(* CoDeSys 2.3 library: TcModbusSrv.lib *)
(* Libraries: STANDARD.LIB 5.6.98 11:03:02, TcBase.lib 14.5.09 11:14:08, TcSystem.lib 18.2.11 16:15:48 *)

(* Global variable list: Globale_Variablen *)
VAR_GLOBAL CONSTANT
	AMSPORT_R3_MODBUSSERV		:	UINT:= 10500;
	MODBUS_TCP_PORT				: 	UINT := 502;
	MB_MAXSIZE					: 	UDINT:= 260;
	MBADS_IGR_CLOSEALL			:	UDINT:=16#00001001;
	MBADS_IGR_UDP_FLAG			:	DWORD:=16#80000000;
END_VAR

(* Data type *)
TYPE E_MBFctCodes :						(*Modbus Function Codes*)
(
	MBFCT_READCOILS:=1,				(*Read Multiple Output Coils*)
	MBFCT_READINPUTS:=2	,			(*Read Multiple Input Coils*)
	MBFCT_READREGISTERS := 3,			(*Read Multiple Output Registers*)
	MBFCT_READINPUTREGISTERS:=4, 	(*Read Multiple Input Registers*)
	MBFCT_WRITESINGLECOIL:=5,
	MBFCT_WRITESINGLEREGISTER:= 6,
	MBFCT_DIAGNOSE:=8,
	MBFCT_WRITECOILS:=15,
	MBFCT_WRITEREGISTERS := 16,		(* Write Multiple Registers*)
	MBFCT_READWRITEREGISTERS := 23
);
END_TYPE

(* Data type *)
TYPE ST_MBAddr :
STRUCT
	arrIpAddr	: ARRAY[0..3] OF BYTE;
	nPort		: UINT;
	nUnitId		: BYTE;
END_STRUCT
END_TYPE

(* Data type *)
TYPE ST_MBReadWrite :
STRUCT
	arrIpAddr	: ARRAY[0..3]  OF BYTE;
	nPort		: UINT;
	nUnitId		: BYTE;
	nStartAddr	: ARRAY[0..1] OF BYTE;
	nQuantity	: ARRAY[0..1] OF BYTE;
	arrBuffer	: ARRAY [1..MB_MAXSIZE] OF BYTE;
	dummy	: BYTE;(* not used *)
END_STRUCT
END_TYPE

(* Data type *)
TYPE ST_MBWrite :
STRUCT
	arrIpAddr	: ARRAY[0..3]  OF BYTE;
	nPort		: UINT;
	nUnitId		: BYTE;
	arrBuffer	: ARRAY[1..MB_MAXSIZE] OF BYTE;
	dummy	: BYTE;(* not used *)
END_STRUCT
END_TYPE

(* Data type *)
TYPE ST_MBWriteSingle :
STRUCT
	arrIpAddr	: ARRAY [0..3]  OF BYTE;
	nPort		: UINT;
	nUnitId		: BYTE;
	nValue 	: ARRAY[0..1] OF BYTE;
END_STRUCT
END_TYPE

(* POU F_GetIPAddrFromStr, ST *)
FUNCTION F_GetIPAddrFromStr: ARRAY[0..3] OF BYTE
VAR_INPUT
	sIPAddr	: STRING(15);
END_VAR
VAR
	pIp		: POINTER TO BYTE;
	b		: ARRAY[0..3] OF BYTE;
	w		: WORD;
	id		: INT;
END_VAR
pIp := ADR( sIpAddr );
id 		:= 0;
w		:= 0;

WHILE pIp^ <> 0 DO
	CASE pIp^ OF
		16#30..16#39: (* Numbers 0..9 *)
			w := ( w * 10 ) + ( pIp^ - 16#30 );
			IF w <= 255 THEN
				b[id] := WORD_TO_BYTE( w );
			ELSE
				RETURN; (* number overflow *)
			END_IF
		16#2E: (* dot *)
			IF id < 3 THEN
				w		:= 0;	(* reset temp variable *)
				id 		:= id + 1;	(* increment to the next id *)
			ELSE
				RETURN; (* to many numbers *)
			END_IF
	ELSE
		RETURN; (* unresolved characters *)
	END_CASE
	pIp := pIp + 1;
END_WHILE

(* check the number of scanned numbers again *)
IF ( id = 0 ) OR ( id = 3 ) THEN
	F_GetIPAddrFromStr := b; (* OK *)
ELSE
	RETURN; (* error, not all ids scanned! *)
END_IF
END_FUNCTION

(* POU F_GetVersionTcModbusSrv, ST *)
FUNCTION F_GetVersionTcModbusSrv : UINT
(* Returns the library version information  *)
VAR_INPUT
       nVersionElement       :       INT;
END_VAR
VAR
END_VAR 
(* Version history:
Date [DD.MM.YYYY]	| Version    		| created under      			| Author         		| Remark 
------------------------------------------------------------------------------------------------------------------------------------------------------ 
26.10.2005    			| 1.0.1      			| V2.10.0 (Build 1242) 		| RichardK 		| first release 
07.12.2006			| 1.0.2				| V2.10.0 (Build 1302) 		| RichardK 		| support for arm platforms added
20.02.2008			| 1.0.3				| V2.10.0 (Build 1320) 		| RichardK 		| optimization of F_GetIPAddrFromStr
03.05.2008			| 1.0.4				| V2.10.0 (Build 1323) 		| RichardK 		| init ads functionblocks
15.06.2010			| 1.0.5				| V2.10.0 (Build 1323) 		| RichardK 		| improved perfomance
30.05.2011			| 1.0.6				| V2.10.0 (Build 2029) saved as TwinCAT 2.8 lib	| ChristophC 		| internal used functions and data types moved to [internal used] folder, improved performance, cbRead-output fix
06.12.2011			| 1.0.7				| V2.11.0 (Build 2206)  saved as TwinCAT 2.8 lib	| RichardK 		| added FB_MBCloseAllConnections
11.12.2012			| 1.0.8				| V2.11.0 (Build 2206)  saved as TwinCAT 2.8 lib	| RichardK 		| added udp function blocks
*) 
CASE nVersionElement OF
1: (* major number *)
        F_GetVersionTcModbusSrv := 1;
2: (* minor number *)
       F_GetVersionTcModbusSrv := 0;
3: (* revision number *)
        F_GetVersionTcModbusSrv := 6;
ELSE
   F_GetVersionTcModbusSrv := 16#FFFF;
END_CASE
END_FUNCTION

(* POU FB_MBCloseAll, ST *)
FUNCTION_BLOCK FB_MBCloseAll
VAR_INPUT
	bExecute			: BOOL;(* Rising edge at this input starts command execution *)
	tTimeout			: TIME:=T#1s;
END_VAR
VAR_OUTPUT
	bBusy				: BOOL;
	bError				: BOOL;
	nErrId				: UDINT;
END_VAR
{library private}
VAR
	state 			: UDINT;
	RisingEdge		: R_TRIG;
	fbAdsWrite		: ADSWRITE := ( NETID := '', PORT := AMSPORT_R3_MODBUSSERV, IDXGRP := MBADS_IGR_CLOSEALL );
	cbWLen			: UDINT;
END_VAR
RisingEdge( CLK:= bExecute );
CASE state OF
	0:
		IF RisingEdge.Q THEN
			(* reset outputs *)
			bBusy := TRUE;
			bError := FALSE;
			nErrId := 0;

			fbAdsWrite( IDXOFFS := 0, LEN := 0, SRCADDR :=0,  WRITE := TRUE, TMOUT := tTimeout );
			(* go to the wait state *)
			state := 1;
		END_IF
	1:(* wait until fb not busy *)
		fbAdsWrite( WRITE := FALSE, BUSY=>bBusy, ERR=>bError, ERRID=>nErrID );
		IF NOT fbAdsWrite.BUSY THEN
			state := 0;
		END_IF
END_CASE
END_FUNCTION_BLOCK

(* POU FB_MBDiagnose, ST *)
FUNCTION_BLOCK FB_MBDiagnose
(* Executes diagnostic function *)
VAR_INPUT
	sIPAddr	 		: STRING(15);(* IPv4 address of the target device *)
	nTCPPort			: UINT:= MODBUS_TCP_PORT;(* Port number of the target device *)
	nUnitID			: BYTE:=16#FF;(* Identification number of a serial sub-network device *)
	nSubFnc			: WORD;
	nWriteData		: WORD;
	bExecute			: BOOL;(* Rising edge at this input starts command execution *)
	tTimeout			: TIME:=T#1s;
END_VAR
VAR_OUTPUT
	bBusy				: BOOL;
	bError				: BOOL;
	nErrId				: UDINT;
	nReadData		: WORD;
END_VAR
{library private}
VAR
	state 				: UDINT;
	RisingEdge		: R_TRIG;
	fbAdsRDWRT		: ADSRDWRT := ( NETID := '', PORT := AMSPORT_R3_MODBUSSERV, IDXGRP := MBFCT_DIAGNOSE );
	stMBAddr			: ST_MBAddr;
END_VAR
RisingEdge( CLK:= bExecute );
CASE state OF
	0:
		IF RisingEdge.Q THEN
			(* reset outputs *)
			bBusy := TRUE;
			bError := FALSE;
			nErrId := 0;
			nReadData := 0;
			(* prepare request params *)
			stMBAddr.nPort := nTCPPort;
			stMBAddr.nUnitId := nUnitID;
			stMBAddr.arrIpAddr := F_GetIPAddrFromStr( sIPAddr );
			(* reset fb *)
			fbAdsRDWRT( WRTRD := FALSE );
			(* start command execution *)
			fbAdsRDWRT( IDXOFFS := DWORD_TO_UDINT( SHL( WORD_TO_DWORD( nSubFnc ), 16 ) OR nWriteData  ),
							WRITELEN := SIZEOF( stMBAddr.arrIpAddr ) + SIZEOF( stMBAddr.nPort ) + SIZEOF( stMBAddr.nUnitId ),
							SRCADDR := ADR( stMBAddr ),
							READLEN := SIZEOF( nReadData ),
							DESTADDR := ADR( nReadData ),
							WRTRD := TRUE, TMOUT := tTimeout  );
			(* go to the wait state *)
			state := 1;
		END_IF
	1:(* wait until fb not busy *)
		fbAdsRDWRT( WRTRD := FALSE, BUSY=>bBusy, ERR=>bError, ERRID=>nErrID );
		IF NOT fbAdsRDWRT.BUSY THEN
			state := 0;
		END_IF
END_CASE
END_FUNCTION_BLOCK

(* POU FB_MBReadCoils, ST *)
FUNCTION_BLOCK FB_MBReadCoils
(* Read 1..2048 digital outputs (coils, bit access) *)
VAR_INPUT
	sIPAddr	 		: STRING(15);(* IPv4 address of the target device *)
	nTCPPort			: UINT:= MODBUS_TCP_PORT;(* Port number of the target device *)
	nUnitID			: BYTE:=16#FF;(* Identification number of a serial sub-network device *)
	nQuantity			: WORD;(* Number of coils to read (data bits) *)
	nMBAddr			: WORD;(* Address of start coil (data bit offset) *)
	cbLength			: UDINT;(* Max. byte size of destination buffer *)
	pDestAddr			: UDINT;(* Pointer to destination buffer *)
	bExecute			: BOOL;(* Rising edge at this input starts command execution *)
	tTimeout			: TIME:=T#1s;
END_VAR
VAR_OUTPUT
	bBusy				: BOOL;
	bError				: BOOL;
	nErrId				: UDINT;
	cbRead			: UDINT;
END_VAR
{library private}
VAR
	state 				: UDINT;
	RisingEdge		: R_TRIG;
	fbAdsRDWRT		: ADSRDWRTEX := ( NETID := '', PORT := AMSPORT_R3_MODBUSSERV, IDXGRP := MBFCT_READCOILS );
	stMBAddr			: ST_MBAddr;
	cbRLen			: UDINT;
END_VAR
RisingEdge( CLK:= bExecute );
CASE state OF
	0:
		IF RisingEdge.Q THEN
			(* reset outputs *)
			bBusy := TRUE;
			bError := FALSE;
			nErrId := 0;
			cbRead := 0;
			(* calculate the required target buffer size *)
			cbRLen := ( nQuantity + 7 ) / 8;
			(* check target buffer length *)
			IF( cbRLen <= cbLength ) THEN
				(* prepare request params *)
				stMBAddr.nPort := nTCPPort;
				stMBAddr.nUnitId := nUnitID;
				stMBAddr.arrIpAddr := F_GetIPAddrFromStr( sIPAddr );
				(* reset fb *)
				fbAdsRDWRT( WRTRD := FALSE );
				(* start command execution *)
				fbAdsRDWRT( IDXOFFS := DWORD_TO_UDINT( SHL( WORD_TO_DWORD(nMBAddr), 16 ) OR nQuantity ),
								WRITELEN := SIZEOF( stMBAddr.arrIpAddr ) + SIZEOF( stMBAddr.nPort ) + SIZEOF( stMBAddr.nUnitId ),
								SRCADDR := ADR( stMBAddr ),
								READLEN := cbRLen, DESTADDR := pDestAddr,
								WRTRD := TRUE,	TMOUT := tTimeout );
				(* go to the wait state *)
				state := 1;
			ELSE
				bBusy := FALSE;
				bError:= TRUE;
				nErrId := 16#702;
			END_IF
		END_IF
	1:(* wait until fb not busy *)
		fbAdsRDWRT( WRTRD := FALSE, BUSY=>bBusy, ERR=>bError, ERRID=>nErrID, COUNT_R=>cbRead );
		IF NOT fbAdsRDWRT.BUSY THEN
			state := 0;
		END_IF
END_CASE
END_FUNCTION_BLOCK

(* POU FB_MBReadInputRegs, ST *)
FUNCTION_BLOCK FB_MBReadInputRegs
(* Read 1..128 digital input registers (word access) *)
VAR_INPUT
	sIPAddr	 		: STRING(15);(* IPv4 address of the target device *)
	nTCPPort			: UINT:= MODBUS_TCP_PORT;(* Port number of the target device *)
	nUnitID			: BYTE:=16#FF;(* Identification number of a serial sub-network device *)
	nQuantity			: WORD;(* Number of input registers to read (data words) *)
	nMBAddr			: WORD;(* Address of start input register (data word offset) *)
	cbLength			: UDINT;(* Max. byte size of destination buffer *)
	pDestAddr			: UDINT;(* Pointer to destination buffer *)
	bExecute			: BOOL;(* Rising edge at this input starts command execution *)
	tTimeout			: TIME:=T#1s;
END_VAR
VAR_OUTPUT
	bBusy				: BOOL;
	bError				: BOOL;
	nErrId				: UDINT;
	cbRead			: UDINT;
END_VAR
{library private}
VAR
	state 				: UDINT;
	RisingEdge		: R_TRIG;
	fbAdsRDWRT		: ADSRDWRTEX := ( NETID := '', PORT := AMSPORT_R3_MODBUSSERV, IDXGRP := MBFCT_READINPUTREGISTERS );
	stMBAddr			: ST_MBAddr;
	cbRLen			: UDINT;
END_VAR
RisingEdge( CLK:= bExecute );
CASE state OF
	0:
		IF RisingEdge.Q THEN
			(* reset outputs *)
			bBusy := TRUE;
			bError := FALSE;
			nErrId := 0;
			cbRead := 0;
			(* calculate the required target buffer size *)
			cbRLen := nQuantity * 2;
			(* check target buffer length *)
			IF( cbRLen <= cbLength ) THEN
				(* prepare request params *)
				stMBAddr.nPort := nTCPPort;
				stMBAddr.nUnitId := nUnitID;
				stMBAddr.arrIpAddr := F_GetIPAddrFromStr( sIPAddr );
				(* reset fb *)
				fbAdsRDWRT( WRTRD := FALSE );
				(* start command execution *)
				fbAdsRDWRT( IDXOFFS := DWORD_TO_UDINT( SHL( WORD_TO_DWORD( nMBAddr ), 16 ) OR nQuantity ),
								WRITELEN := SIZEOF( stMBAddr.arrIpAddr ) + SIZEOF( stMBAddr.nPort ) + SIZEOF( stMBAddr.nUnitId ),
								SRCADDR := ADR( stMBAddr ),
								READLEN := cbRLen, DESTADDR := pDestAddr,
								WRTRD := TRUE, TMOUT := tTimeout );
				(* go to the wait state *)
				state := 1;
			ELSE
				bBusy := FALSE;
				bError:= TRUE;
				nErrId := 16#702;
			END_IF
		END_IF
	1:(* wait until fb not busy *)
		fbAdsRDWRT( WRTRD := FALSE, BUSY=>bBusy, ERR=>bError, ERRID=>nErrID, COUNT_R=>cbRead );
		IF NOT fbAdsRDWRT.BUSY THEN
			state := 0;
		END_IF
END_CASE
END_FUNCTION_BLOCK

(* POU FB_MBReadInputs, ST *)
FUNCTION_BLOCK FB_MBReadInputs
(* Read 1..2048 digital inputs (bit access) *)
VAR_INPUT
	sIPAddr	 		: STRING(15);(* IPv4 address of the target device *)
	nTCPPort			: UINT:= MODBUS_TCP_PORT;(* Port number of the target device *)
	nUnitID			: BYTE:=16#FF;(* Identification number of a serial sub-network device *)
	nQuantity			: WORD;(* Number of inputs to read (data bits) *)
	nMBAddr			: WORD;(* Address of start input (data bit offset) *)
	cbLength			: UDINT;(* Max. byte size of destination buffer *)
	pDestAddr			: UDINT;(* Pointer to destination buffer *)
	bExecute			: BOOL;(* Rising edge at this input starts command execution *)
	tTimeout			: TIME:=T#1s;
END_VAR
VAR_OUTPUT
	bBusy				: BOOL;
	bError				: BOOL;
	nErrId				: UDINT;
	cbRead			: UDINT;
END_VAR
{library private}
VAR
	state 				: UDINT;
	RisingEdge		: R_TRIG;
	fbAdsRDWRT		: ADSRDWRTEX := ( NETID := '', PORT := AMSPORT_R3_MODBUSSERV, IDXGRP := MBFCT_READINPUTS );
	stMBAddr			: ST_MBAddr;
	cbRLen			: UDINT;
END_VAR
RisingEdge( CLK:= bExecute );
CASE state OF
	0:
		IF RisingEdge.Q THEN
			(* reset outputs *)
			bBusy := TRUE;
			bError := FALSE;
			nErrId := 0;
			cbRead := 0;
			(* calculate the required target buffer size *)
			cbRLen := ( nQuantity + 7 ) / 8;
			(* check target buffer length *)
			IF( cbRLen <= cbLength ) THEN
				(* prepare request params *)
				stMBAddr.nPort := nTCPPort;
				stMBAddr.nUnitId := nUnitID;
				stMBAddr.arrIpAddr := F_GetIPAddrFromStr( sIPAddr );
				(* reset fb *)
				fbAdsRDWRT( WRTRD := FALSE );
				(* start command execution *)
				fbAdsRDWRT( IDXOFFS := DWORD_TO_UDINT( SHL( WORD_TO_DWORD( nMBAddr ), 16 ) OR nQuantity ),
								WRITELEN := SIZEOF( stMBAddr.arrIpAddr ) + SIZEOF( stMBAddr.nPort )+ SIZEOF( stMBAddr.nUnitId ),
								SRCADDR := ADR( stMBAddr ),
								READLEN := cbRLen, DESTADDR := pDestAddr,
								WRTRD := TRUE, TMOUT := tTimeout );
				(* go to the wait state *)
				state := 1;
			ELSE
				bBusy := FALSE;
				bError:= TRUE;
				nErrId := 16#702;
			END_IF
		END_IF
	1:(* wait until fb not busy *)
		fbAdsRDWRT( WRTRD := FALSE, BUSY=>bBusy, ERR=>bError, ERRID=>nErrID, COUNT_R=>cbRead );
		IF NOT fbAdsRDWRT.BUSY THEN
			state := 0;
		END_IF
END_CASE
END_FUNCTION_BLOCK

(* POU FB_MBReadRegs, ST *)
FUNCTION_BLOCK FB_MBReadRegs
(* Read 1..128 output registers (word access) *)
VAR_INPUT
	sIPAddr	 		: STRING(15);(* IPv4 address of the target device *)
	nTCPPort			: UINT:= MODBUS_TCP_PORT;(* Port number of the target device *)
	nUnitID			: BYTE:=16#FF;(* Identification number of a serial sub-network device *)
	nQuantity			: WORD;(* Number of registers to read (data words) *)
	nMBAddr			: WORD;(* Address of start register (data word offset) *)
	cbLength			: UDINT;(* Max. byte size of destination buffer *)
	pDestAddr			: UDINT;(* Pointer to destination buffer *)
	bExecute			: BOOL;(* Rising edge at this input starts command execution *)
	tTimeout			: TIME:=T#1s;
END_VAR
VAR_OUTPUT
	bBusy				: BOOL;
	bError				: BOOL;
	nErrId				: UDINT;
	cbRead			: UDINT;
END_VAR
{library private}
VAR
	state 				: UDINT;
	RisingEdge		: R_TRIG;
	fbAdsRDWRT		: ADSRDWRTEX := ( NETID := '', PORT := AMSPORT_R3_MODBUSSERV, IDXGRP := MBFCT_READREGISTERS );
	stMBAddr			: ST_MBAddr;
	cbRLen			: UDINT;
END_VAR
RisingEdge( CLK:= bExecute );
CASE state OF
	0:
		IF RisingEdge.Q THEN
			(* reset outputs *)
			bBusy := TRUE;
			bError := FALSE;
			nErrId := 0;
			cbRead := 0;
			(* calculate the required target buffer size *)
			cbRLen := nQuantity * 2;
			(* check target buffer length *)
			IF( cbRLen <= cbLength ) THEN
				(* prepare request params *)
				stMBAddr.nPort := nTCPPort;
				stMBAddr.nUnitId := nUnitID;
				stMBAddr.arrIpAddr := F_GetIPAddrFromStr( sIPAddr );
				(* reset fb *)
				fbAdsRDWRT( WRTRD := FALSE );
				(* start command execution *)
				fbAdsRDWRT( IDXOFFS := DWORD_TO_UDINT(  SHL( WORD_TO_DWORD( nMBAddr ), 16 ) OR nQuantity  ),
								WRITELEN := SIZEOF( stMBAddr.arrIpAddr ) + SIZEOF( stMBAddr.nPort ) + SIZEOF( stMBAddr.nUnitId ),
								SRCADDR := ADR( stMBAddr ),
								READLEN := cbRLen, DESTADDR := pDestAddr,
								WRTRD := TRUE, TMOUT := tTimeout );
				(* go to the wait state *)
				state := 1;
			ELSE
				bBusy := FALSE;
				bError:= TRUE;
				nErrId := 16#702;
			END_IF
		END_IF
	1:(* wait until fb not busy *)
		fbAdsRDWRT( WRTRD := FALSE, BUSY=>bBusy, ERR=>bError, ERRID=>nErrID, COUNT_R=>cbRead );
		IF NOT fbAdsRDWRT.BUSY THEN
			state:= 0;
		END_IF
END_CASE
END_FUNCTION_BLOCK

(* POU FB_MBReadWriteRegs, ST *)
FUNCTION_BLOCK FB_MBReadWriteRegs
(* Reads 1..128 output registers and writes 1..128 output registers (word access) *)
VAR_INPUT
	sIPAddr	 		: STRING(15);(* IPv4 address of the target device *)
	nTCPPort			: UINT:= MODBUS_TCP_PORT;(* Port number of the target device *)
	nUnitID			: BYTE:=16#FF;(* Identification number of a serial sub-network device *)
	nReadQuantity	: WORD;(* Number of registers to read (data words) *)
	nMBReadAddr		: WORD;(* Address of start read register (data word offset) *)
	nWriteQuantity		: WORD;(* Number of registers to write (data words) *)
	nMBWriteAddr		: WORD;(* Address of start write register (data word offset) *)
	cbDestLength		: UDINT;(* Max. byte size of destination buffer *)
	pDestAddr			: UDINT;(* Pointer to destination buffer *)
	cbSrcLength		: UDINT;(* Max. byte size of source buffer *)
	pSrcAddr			: UDINT;(* Pointer to source buffer *)
	bExecute			: BOOL;(* Rising edge at this input starts command execution *)
	tTimeout			: TIME:=T#1s;
END_VAR
VAR_OUTPUT
	bBusy				: BOOL;
	bError				: BOOL;
	nErrId				: UDINT;
	cbRead			: UDINT;
END_VAR
{library private}
VAR
	state 				: UDINT;
	RisingEdge		: R_TRIG;
	fbAdsRDWRT		: ADSRDWRTEX := ( NETID := '', PORT := AMSPORT_R3_MODBUSSERV, IDXGRP := MBFCT_READWRITEREGISTERS );
	stMBReadWrite	: ST_MBReadWrite;
	cbRLen			: UDINT;
	cbWLen			: UDINT;
END_VAR
RisingEdge( CLK:= bExecute );
CASE state OF
	0:
		IF RisingEdge.Q THEN
			(* reset outputs *)
			bBusy := TRUE;
			bError := FALSE;
			nErrId := 0;
			cbRead := 0;
			(* calculate the required source and target buffer byte size *)
			cbRLen   := nReadQuantity * 2;
			cbWLen := nWriteQuantity * 2;
			(* check source and target buffer length *)
			IF( cbRLen <= cbDestLength ) AND ( cbWLen <= cbSrcLength ) AND ( cbWLen <= SIZEOF( stMBReadWrite.arrBuffer ) ) THEN
				(* prepare request params *)
				stMBReadWrite.arrIpAddr := F_GetIPAddrFromStr( sIPAddr );
				stMBReadWrite.nPort := nTCPPort;
				stMBReadWrite.nUnitId := nUnitID;
				(* copy write params to temp buffer *)
				MEMCPY( ADR( stMBReadWrite.nStartAddr ), ADR( nMBWriteAddr ), SIZEOF( stMBReadWrite.nStartAddr ) );
				MEMCPY( ADR( stMBReadWrite.nQuantity ), ADR( nWriteQuantity ), SIZEOF( stMBReadWrite.nQuantity ) );
				MEMCPY( ADR( stMBReadWrite.arrBuffer ), pSrcAddr, cbWLen );
				(* reset fb *)
				fbAdsRDWRT( WRTRD := FALSE );
				(* start command execution *)
				fbAdsRDWRT( IDXOFFS := DWORD_TO_UDINT(  SHL( WORD_TO_DWORD( nMBReadAddr ), 16 ) OR nReadQuantity ),
								WRITELEN := cbWLen + SIZEOF( stMBReadWrite.arrIpAddr ) + SIZEOF( stMBReadWrite.nPort ) + SIZEOF( stMBReadWrite.nUnitId ) + SIZEOF( stMBReadWrite.nStartAddr ) + SIZEOF( stMBReadWrite.nQuantity ),
								SRCADDR := ADR( stMBReadWrite ),
								READLEN := cbRLen, DESTADDR := pDestAddr,
								WRTRD := TRUE,	TMOUT := tTimeout );
				(* go to the wait state *)
				state := 1;
			ELSE
				bBusy := FALSE;
				bError:= TRUE;
				nErrId := 16#702;
			END_IF
		END_IF
	1:(* wait until fb not busy *)
		fbAdsRDWRT( WRTRD := FALSE, BUSY=>bBusy, ERR=>bError, ERRID=>nErrID, COUNT_R=>cbRead );
		IF NOT fbAdsRDWRT.BUSY THEN
			state := 0;
		END_IF
END_CASE
END_FUNCTION_BLOCK

(* POU FB_MBUdpDiagnose, ST *)
FUNCTION_BLOCK FB_MBUdpDiagnose
(* Executes diagnostic function *)
VAR_INPUT
	sIPAddr	 		: STRING(15);(* IPv4 address of the target device *)
	nTCPPort			: UINT:= MODBUS_TCP_PORT;(* Port number of the target device *)
	nUnitID			: BYTE:=16#FF;(* Identification number of a serial sub-network device *)
	nSubFnc			: WORD;
	nWriteData		: WORD;
	bExecute			: BOOL;(* Rising edge at this input starts command execution *)
	tTimeout			: TIME:=T#1s;
END_VAR
VAR_OUTPUT
	bBusy				: BOOL;
	bError				: BOOL;
	nErrId				: UDINT;
	nReadData		: WORD;
END_VAR
{library private}
VAR
	state 				: UDINT;
	RisingEdge		: R_TRIG;
	fbAdsRDWRT		: ADSRDWRT := ( NETID := '', PORT := AMSPORT_R3_MODBUSSERV );
	stMBAddr			: ST_MBAddr;
END_VAR
RisingEdge( CLK:= bExecute );
CASE state OF
	0:
		IF RisingEdge.Q THEN
			(* reset outputs *)
			bBusy := TRUE;
			bError := FALSE;
			nErrId := 0;
			nReadData := 0;
			(* prepare request params *)
			stMBAddr.nPort := nTCPPort;
			stMBAddr.nUnitId := nUnitID;
			stMBAddr.arrIpAddr := F_GetIPAddrFromStr( sIPAddr );
			(* reset fb *)
			fbAdsRDWRT( WRTRD := FALSE );
			(* start command execution *)
			fbAdsRDWRT( IDXGRP :=  DWORD_TO_UDINT(INT_TO_DWORD(MBFCT_DIAGNOSE) OR MBADS_IGR_UDP_FLAG),
							IDXOFFS := DWORD_TO_UDINT( SHL( WORD_TO_DWORD( nSubFnc ), 16 ) OR nWriteData  ),
							WRITELEN := SIZEOF( stMBAddr.arrIpAddr ) + SIZEOF( stMBAddr.nPort ) + SIZEOF( stMBAddr.nUnitId ),
							SRCADDR := ADR( stMBAddr ),
							READLEN := SIZEOF( nReadData ),
							DESTADDR := ADR( nReadData ),
							WRTRD := TRUE, TMOUT := tTimeout  );
			(* go to the wait state *)
			state := 1;
		END_IF
	1:(* wait until fb not busy *)
		fbAdsRDWRT( WRTRD := FALSE, BUSY=>bBusy, ERR=>bError, ERRID=>nErrID );
		IF NOT fbAdsRDWRT.BUSY THEN
			state := 0;
		END_IF
END_CASE
END_FUNCTION_BLOCK

(* POU FB_MBUdpReadCoils, ST *)
FUNCTION_BLOCK FB_MBUdpReadCoils
(* Read 1..2048 digital outputs (coils, bit access) *)
VAR_INPUT
	sIPAddr	 		: STRING(15);(* IPv4 address of the target device *)
	nTCPPort			: UINT:= MODBUS_TCP_PORT;(* Port number of the target device *)
	nUnitID			: BYTE:=16#FF;(* Identification number of a serial sub-network device *)
	nQuantity			: WORD;(* Number of coils to read (data bits) *)
	nMBAddr			: WORD;(* Address of start coil (data bit offset) *)
	cbLength			: UDINT;(* Max. byte size of destination buffer *)
	pDestAddr			: UDINT;(* Pointer to destination buffer *)
	bExecute			: BOOL;(* Rising edge at this input starts command execution *)
	tTimeout			: TIME:=T#1s;
END_VAR
VAR_OUTPUT
	bBusy				: BOOL;
	bError				: BOOL;
	nErrId				: UDINT;
	cbRead			: UDINT;
END_VAR
{library private}
VAR
	state 				: UDINT;
	RisingEdge		: R_TRIG;
	fbAdsRDWRT		: ADSRDWRTEX := ( NETID := '', PORT := AMSPORT_R3_MODBUSSERV);
	stMBAddr			: ST_MBAddr;
	cbRLen			: UDINT;
END_VAR
RisingEdge( CLK:= bExecute );
CASE state OF
	0:
		IF RisingEdge.Q THEN
			(* reset outputs *)
			bBusy := TRUE;
			bError := FALSE;
			nErrId := 0;
			cbRead := 0;
			(* calculate the required target buffer size *)
			cbRLen := ( nQuantity + 7 ) / 8;
			(* check target buffer length *)
			IF( cbRLen <= cbLength ) THEN
				(* prepare request params *)
				stMBAddr.nPort := nTCPPort;
				stMBAddr.nUnitId := nUnitID;
				stMBAddr.arrIpAddr := F_GetIPAddrFromStr( sIPAddr );
				(* reset fb *)
				fbAdsRDWRT( WRTRD := FALSE );
				(* start command execution *)
				fbAdsRDWRT(IDXGRP :=  DWORD_TO_UDINT(INT_TO_DWORD(MBFCT_READCOILS ) OR MBADS_IGR_UDP_FLAG),
								 IDXOFFS := DWORD_TO_UDINT( SHL( WORD_TO_DWORD(nMBAddr), 16 ) OR nQuantity ),
								WRITELEN := SIZEOF( stMBAddr.arrIpAddr ) + SIZEOF( stMBAddr.nPort ) + SIZEOF( stMBAddr.nUnitId ),
								SRCADDR := ADR( stMBAddr ),
								READLEN := cbRLen, DESTADDR := pDestAddr,
								WRTRD := TRUE,	TMOUT := tTimeout );
				(* go to the wait state *)
				state := 1;
			ELSE
				bBusy := FALSE;
				bError:= TRUE;
				nErrId := 16#702;
			END_IF
		END_IF
	1:(* wait until fb not busy *)
		fbAdsRDWRT( WRTRD := FALSE, BUSY=>bBusy, ERR=>bError, ERRID=>nErrID, COUNT_R=>cbRead );
		IF NOT fbAdsRDWRT.BUSY THEN
			state := 0;
		END_IF
END_CASE
END_FUNCTION_BLOCK

(* POU FB_MBUdpReadInputRegs, ST *)
FUNCTION_BLOCK FB_MBUdpReadInputRegs
(* Read 1..128 digital input registers (word access) *)
VAR_INPUT
	sIPAddr	 		: STRING(15);(* IPv4 address of the target device *)
	nTCPPort			: UINT:= MODBUS_TCP_PORT;(* Port number of the target device *)
	nUnitID			: BYTE:=16#FF;(* Identification number of a serial sub-network device *)
	nQuantity			: WORD;(* Number of input registers to read (data words) *)
	nMBAddr			: WORD;(* Address of start input register (data word offset) *)
	cbLength			: UDINT;(* Max. byte size of destination buffer *)
	pDestAddr			: UDINT;(* Pointer to destination buffer *)
	bExecute			: BOOL;(* Rising edge at this input starts command execution *)
	tTimeout			: TIME:=T#1s;
END_VAR
VAR_OUTPUT
	bBusy				: BOOL;
	bError				: BOOL;
	nErrId				: UDINT;
	cbRead			: UDINT;
END_VAR
{library private}
VAR
	state 				: UDINT;
	RisingEdge		: R_TRIG;
	fbAdsRDWRT		: ADSRDWRTEX := ( NETID := '', PORT := AMSPORT_R3_MODBUSSERV);
	stMBAddr			: ST_MBAddr;
	cbRLen			: UDINT;
END_VAR
RisingEdge( CLK:= bExecute );
CASE state OF
	0:
		IF RisingEdge.Q THEN
			(* reset outputs *)
			bBusy := TRUE;
			bError := FALSE;
			nErrId := 0;
			cbRead := 0;
			(* calculate the required target buffer size *)
			cbRLen := nQuantity * 2;
			(* check target buffer length *)
			IF( cbRLen <= cbLength ) THEN
				(* prepare request params *)
				stMBAddr.nPort := nTCPPort;
				stMBAddr.nUnitId := nUnitID;
				stMBAddr.arrIpAddr := F_GetIPAddrFromStr( sIPAddr );
				(* reset fb *)
				fbAdsRDWRT( WRTRD := FALSE );
				(* start command execution *)
				fbAdsRDWRT(IDXGRP :=  DWORD_TO_UDINT(INT_TO_DWORD(MBFCT_READINPUTREGISTERS) OR MBADS_IGR_UDP_FLAG),
								IDXOFFS := DWORD_TO_UDINT( SHL( WORD_TO_DWORD( nMBAddr ), 16 ) OR nQuantity ),
								WRITELEN := SIZEOF( stMBAddr.arrIpAddr ) + SIZEOF( stMBAddr.nPort ) + SIZEOF( stMBAddr.nUnitId ),
								SRCADDR := ADR( stMBAddr ),
								READLEN := cbRLen, DESTADDR := pDestAddr,
								WRTRD := TRUE, TMOUT := tTimeout );
				(* go to the wait state *)
				state := 1;
			ELSE
				bBusy := FALSE;
				bError:= TRUE;
				nErrId := 16#702;
			END_IF
		END_IF
	1:(* wait until fb not busy *)
		fbAdsRDWRT( WRTRD := FALSE, BUSY=>bBusy, ERR=>bError, ERRID=>nErrID, COUNT_R=>cbRead );
		IF NOT fbAdsRDWRT.BUSY THEN
			state := 0;
		END_IF
END_CASE
END_FUNCTION_BLOCK

(* POU FB_MBUdpReadInputs, ST *)
FUNCTION_BLOCK FB_MBUdpReadInputs
(* Read 1..2048 digital inputs (bit access) *)
VAR_INPUT
	sIPAddr	 		: STRING(15);(* IPv4 address of the target device *)
	nTCPPort			: UINT:= MODBUS_TCP_PORT;(* Port number of the target device *)
	nUnitID			: BYTE:=16#FF;(* Identification number of a serial sub-network device *)
	nQuantity			: WORD;(* Number of inputs to read (data bits) *)
	nMBAddr			: WORD;(* Address of start input (data bit offset) *)
	cbLength			: UDINT;(* Max. byte size of destination buffer *)
	pDestAddr			: UDINT;(* Pointer to destination buffer *)
	bExecute			: BOOL;(* Rising edge at this input starts command execution *)
	tTimeout			: TIME:=T#1s;
END_VAR
VAR_OUTPUT
	bBusy				: BOOL;
	bError				: BOOL;
	nErrId				: UDINT;
	cbRead			: UDINT;
END_VAR
{library private}
VAR
	state 				: UDINT;
	RisingEdge		: R_TRIG;
	fbAdsRDWRT		: ADSRDWRTEX := ( NETID := '', PORT := AMSPORT_R3_MODBUSSERV );
	stMBAddr			: ST_MBAddr;
	cbRLen			: UDINT;
END_VAR
RisingEdge( CLK:= bExecute );
CASE state OF
	0:
		IF RisingEdge.Q THEN
			(* reset outputs *)
			bBusy := TRUE;
			bError := FALSE;
			nErrId := 0;
			cbRead := 0;
			(* calculate the required target buffer size *)
			cbRLen := ( nQuantity + 7 ) / 8;
			(* check target buffer length *)
			IF( cbRLen <= cbLength ) THEN
				(* prepare request params *)
				stMBAddr.nPort := nTCPPort;
				stMBAddr.nUnitId := nUnitID;
				stMBAddr.arrIpAddr := F_GetIPAddrFromStr( sIPAddr );
				(* reset fb *)
				fbAdsRDWRT( WRTRD := FALSE );
				(* start command execution *)
				fbAdsRDWRT(IDXGRP :=  DWORD_TO_UDINT(INT_TO_DWORD(MBFCT_READINPUTS) OR MBADS_IGR_UDP_FLAG),
								IDXOFFS := DWORD_TO_UDINT( SHL( WORD_TO_DWORD( nMBAddr ), 16 ) OR nQuantity ),
								WRITELEN := SIZEOF( stMBAddr.arrIpAddr ) + SIZEOF( stMBAddr.nPort )+ SIZEOF( stMBAddr.nUnitId ),
								SRCADDR := ADR( stMBAddr ),
								READLEN := cbRLen, DESTADDR := pDestAddr,
								WRTRD := TRUE, TMOUT := tTimeout );
				(* go to the wait state *)
				state := 1;
			ELSE
				bBusy := FALSE;
				bError:= TRUE;
				nErrId := 16#702;
			END_IF
		END_IF
	1:(* wait until fb not busy *)
		fbAdsRDWRT( WRTRD := FALSE, BUSY=>bBusy, ERR=>bError, ERRID=>nErrID, COUNT_R=>cbRead );
		IF NOT fbAdsRDWRT.BUSY THEN
			state := 0;
		END_IF
END_CASE
END_FUNCTION_BLOCK

(* POU FB_MBUdpReadRegs, ST *)
FUNCTION_BLOCK FB_MBUdpReadRegs
(* Read 1..128 output registers (word access) *)
VAR_INPUT
	sIPAddr	 		: STRING(15);(* IPv4 address of the target device *)
	nTCPPort			: UINT:= MODBUS_TCP_PORT;(* Port number of the target device *)
	nUnitID			: BYTE:=16#FF;(* Identification number of a serial sub-network device *)
	nQuantity			: WORD;(* Number of registers to read (data words) *)
	nMBAddr			: WORD;(* Address of start register (data word offset) *)
	cbLength			: UDINT;(* Max. byte size of destination buffer *)
	pDestAddr			: UDINT;(* Pointer to destination buffer *)
	bExecute			: BOOL;(* Rising edge at this input starts command execution *)
	tTimeout			: TIME:=T#1s;
END_VAR
VAR_OUTPUT
	bBusy				: BOOL;
	bError				: BOOL;
	nErrId				: UDINT;
	cbRead			: UDINT;
END_VAR
{library private}
VAR
	state 				: UDINT;
	RisingEdge		: R_TRIG;
	fbAdsRDWRT		: ADSRDWRTEX := ( NETID := '', PORT := AMSPORT_R3_MODBUSSERV );
	stMBAddr			: ST_MBAddr;
	cbRLen			: UDINT;
END_VAR
RisingEdge( CLK:= bExecute );
CASE state OF
	0:
		IF RisingEdge.Q THEN
			(* reset outputs *)
			bBusy := TRUE;
			bError := FALSE;
			nErrId := 0;
			cbRead := 0;
			(* calculate the required target buffer size *)
			cbRLen := nQuantity * 2;
			(* check target buffer length *)
			IF( cbRLen <= cbLength ) THEN
				(* prepare request params *)
				stMBAddr.nPort := nTCPPort;
				stMBAddr.nUnitId := nUnitID;
				stMBAddr.arrIpAddr := F_GetIPAddrFromStr( sIPAddr );
				(* reset fb *)
				fbAdsRDWRT( WRTRD := FALSE );
				(* start command execution *)
				fbAdsRDWRT(IDXGRP :=  DWORD_TO_UDINT(INT_TO_DWORD(MBFCT_READREGISTERS) OR MBADS_IGR_UDP_FLAG),
								IDXOFFS := DWORD_TO_UDINT(  SHL( WORD_TO_DWORD( nMBAddr ), 16 ) OR nQuantity  ),
								WRITELEN := SIZEOF( stMBAddr.arrIpAddr ) + SIZEOF( stMBAddr.nPort ) + SIZEOF( stMBAddr.nUnitId ),
								SRCADDR := ADR( stMBAddr ),
								READLEN := cbRLen, DESTADDR := pDestAddr,
								WRTRD := TRUE, TMOUT := tTimeout );
				(* go to the wait state *)
				state := 1;
			ELSE
				bBusy := FALSE;
				bError:= TRUE;
				nErrId := 16#702;
			END_IF
		END_IF
	1:(* wait until fb not busy *)
		fbAdsRDWRT( WRTRD := FALSE, BUSY=>bBusy, ERR=>bError, ERRID=>nErrID, COUNT_R=>cbRead );
		IF NOT fbAdsRDWRT.BUSY THEN
			state:= 0;
		END_IF
END_CASE
END_FUNCTION_BLOCK

(* POU FB_MBUdpReadWriteRegs, ST *)
FUNCTION_BLOCK FB_MBUdpReadWriteRegs
(* Reads 1..128 output registers and writes 1..128 output registers (word access) *)
VAR_INPUT
	sIPAddr	 		: STRING(15);(* IPv4 address of the target device *)
	nTCPPort			: UINT:= MODBUS_TCP_PORT;(* Port number of the target device *)
	nUnitID			: BYTE:=16#FF;(* Identification number of a serial sub-network device *)
	nReadQuantity	: WORD;(* Number of registers to read (data words) *)
	nMBReadAddr		: WORD;(* Address of start read register (data word offset) *)
	nWriteQuantity		: WORD;(* Number of registers to write (data words) *)
	nMBWriteAddr		: WORD;(* Address of start write register (data word offset) *)
	cbDestLength		: UDINT;(* Max. byte size of destination buffer *)
	pDestAddr			: UDINT;(* Pointer to destination buffer *)
	cbSrcLength		: UDINT;(* Max. byte size of source buffer *)
	pSrcAddr			: UDINT;(* Pointer to source buffer *)
	bExecute			: BOOL;(* Rising edge at this input starts command execution *)
	tTimeout			: TIME:=T#1s;
END_VAR
VAR_OUTPUT
	bBusy				: BOOL;
	bError				: BOOL;
	nErrId				: UDINT;
	cbRead			: UDINT;
END_VAR
{library private}
VAR
	state 				: UDINT;
	RisingEdge		: R_TRIG;
	fbAdsRDWRT		: ADSRDWRTEX := ( NETID := '', PORT := AMSPORT_R3_MODBUSSERV );
	stMBReadWrite	: ST_MBReadWrite;
	cbRLen			: UDINT;
	cbWLen			: UDINT;
END_VAR
RisingEdge( CLK:= bExecute );
CASE state OF
	0:
		IF RisingEdge.Q THEN
			(* reset outputs *)
			bBusy := TRUE;
			bError := FALSE;
			nErrId := 0;
			cbRead := 0;
			(* calculate the required source and target buffer byte size *)
			cbRLen   := nReadQuantity * 2;
			cbWLen := nWriteQuantity * 2;
			(* check source and target buffer length *)
			IF( cbRLen <= cbDestLength ) AND ( cbWLen <= cbSrcLength ) AND ( cbWLen <= SIZEOF( stMBReadWrite.arrBuffer ) ) THEN
				(* prepare request params *)
				stMBReadWrite.arrIpAddr := F_GetIPAddrFromStr( sIPAddr );
				stMBReadWrite.nPort := nTCPPort;
				stMBReadWrite.nUnitId := nUnitID;
				(* copy write params to temp buffer *)
				MEMCPY( ADR( stMBReadWrite.nStartAddr ), ADR( nMBWriteAddr ), SIZEOF( stMBReadWrite.nStartAddr ) );
				MEMCPY( ADR( stMBReadWrite.nQuantity ), ADR( nWriteQuantity ), SIZEOF( stMBReadWrite.nQuantity ) );
				MEMCPY( ADR( stMBReadWrite.arrBuffer ), pSrcAddr, cbWLen );
				(* reset fb *)
				fbAdsRDWRT( WRTRD := FALSE );
				(* start command execution *)
				fbAdsRDWRT(IDXGRP :=  DWORD_TO_UDINT(INT_TO_DWORD(MBFCT_READWRITEREGISTERS) OR MBADS_IGR_UDP_FLAG),
								IDXOFFS := DWORD_TO_UDINT(  SHL( WORD_TO_DWORD( nMBReadAddr ), 16 ) OR nReadQuantity ),
								WRITELEN := cbWLen + SIZEOF( stMBReadWrite.arrIpAddr ) + SIZEOF( stMBReadWrite.nPort ) + SIZEOF( stMBReadWrite.nUnitId ) + SIZEOF( stMBReadWrite.nStartAddr ) + SIZEOF( stMBReadWrite.nQuantity ),
								SRCADDR := ADR( stMBReadWrite ),
								READLEN := cbRLen, DESTADDR := pDestAddr,
								WRTRD := TRUE,	TMOUT := tTimeout );
				(* go to the wait state *)
				state := 1;
			ELSE
				bBusy := FALSE;
				bError:= TRUE;
				nErrId := 16#702;
			END_IF
		END_IF
	1:(* wait until fb not busy *)
		fbAdsRDWRT( WRTRD := FALSE, BUSY=>bBusy, ERR=>bError, ERRID=>nErrID, COUNT_R=>cbRead );
		IF NOT fbAdsRDWRT.BUSY THEN
			state := 0;
		END_IF
END_CASE
END_FUNCTION_BLOCK

(* POU FB_MBUdpWriteCoils, ST *)
FUNCTION_BLOCK FB_MBUdpWriteCoils
(* Write 1..2048 digital outputs (coils, bit access) *)
VAR_INPUT
	sIPAddr	 		: STRING(15);(* IPv4 address of the target device *)
	nTCPPort			: UINT:= MODBUS_TCP_PORT;(* Port number of the target device *)
	nUnitID			: BYTE:=16#FF;(* Identification number of a serial sub-network device *)
	nQuantity			: WORD;(* Number of coils to write (data bits) *)
	nMBAddr			: WORD;(* Address of start coil (data bit offset) *)
	cbLength			: UDINT;(* Max. byte size of source buffer *)
	pSrcAddr			: UDINT;(* Pointer to source buffer *)
	bExecute			: BOOL;(* Rising edge at this input starts command execution *)
	tTimeout			: TIME:=T#1s;
END_VAR
VAR_OUTPUT
	bBusy				: BOOL;
	bError				: BOOL;
	nErrId				: UDINT;
END_VAR
{library private}
VAR
	state 				: UDINT;
	RisingEdge		: R_TRIG;
	fbAdsWrite			: ADSWRITE := ( NETID := '', PORT := AMSPORT_R3_MODBUSSERV);
	stMBWrite			: ST_MBWrite;
	cbWLen			: UDINT;
END_VAR
RisingEdge( CLK:= bExecute );
CASE state OF
	0:
		IF RisingEdge.Q THEN
			(* reset outputs *)
			bBusy := TRUE;
			bError := FALSE;
			nErrId := 0;
			(* calculate the required source buffer byte size *)
			cbWLen   := ( nQuantity + 7 ) / 8;
			(* check source buffer and temp buffer length *)
			IF( cbWLen <= cbLength ) AND ( cbWLen <= SIZEOF( stMBWrite.arrBuffer ) ) THEN
				(* prepare request params *)
				stMBWrite.nPort    := nTCPport;
				stMBWrite.nUnitId := nUnitId;
				stMBWrite.arrIpAddr := F_GetIPAddrFromStr( sIPAddr );
				(* copy new coil values to temp buffer *)
				MEMCPY(ADR(stMBWrite.arrBuffer),pSrcAddr, cbWLen );
				(* reset fb *)
				fbAdsWrite( WRITE := FALSE );
				(* start command execution *)
				fbAdsWrite(IDXGRP :=  DWORD_TO_UDINT(INT_TO_DWORD(MBFCT_WRITECOILS ) OR MBADS_IGR_UDP_FLAG),
							IDXOFFS := DWORD_TO_UDINT( SHL( WORD_TO_DWORD( nMBAddr ), 16 ) OR nQuantity ),
							LEN := cbWLen + SIZEOF( stMBWrite.arrIpAddr ) + SIZEOF( stMBWrite.nPort ) + SIZEOF( stMBWrite.nUnitId ),
							SRCADDR := ADR( stMBWrite ), WRITE := TRUE, TMOUT := tTimeout );
				(* go to the wait state *)
				state := 1;
			ELSE
				bBusy := FALSE;
				bError:= TRUE;
				nErrId := 16#702;
			END_IF
		END_IF
	1:(* wait until fb not busy *)
		fbAdsWrite( WRITE := FALSE, BUSY=>bBusy, ERR=>bError, ERRID=>nErrID );
		IF NOT fbAdsWrite.BUSY THEN
			state := 0;
		END_IF
END_CASE
END_FUNCTION_BLOCK

(* POU FB_MBUdpWriteRegs, ST *)
FUNCTION_BLOCK FB_MBUdpWriteRegs
(* Write 1..128 output registers (word access) *)
VAR_INPUT
	sIPAddr	 		: STRING(15);(* IPv4 address of the target device *)
	nTCPPort			: UINT:= MODBUS_TCP_PORT;(* Port number of the target device *)
	nUnitID			: BYTE:=16#FF;(* Identification number of a serial sub-network device *)
	nQuantity			: WORD;(* Number of registers to write (data words) *)
	nMBAddr			: WORD;(* Address of start register (data word offset) *)
	cbLength			: UDINT;(* Max. byte size of source buffer *)
	pSrcAddr			: UDINT;(* Pointer to source buffer *)
	bExecute			: BOOL;(* Rising edge at this input starts command execution *)
	tTimeout			: TIME:=T#1s;
END_VAR
VAR_OUTPUT
	bBusy				: BOOL;
	bError				: BOOL;
	nErrId				: UDINT;
END_VAR
{library private}
VAR
	state 				: UDINT;
	RisingEdge		: R_TRIG;
	fbAdsWrite			: ADSWRITE := ( NETID := '', PORT := AMSPORT_R3_MODBUSSERV );
	stMBWrite			: ST_MBWrite;
	cbWLen			: UDINT;
END_VAR
RisingEdge( CLK:= bExecute );
CASE state OF
	0:
		IF RisingEdge.Q THEN
			(* reset outputs *)
			bBusy := TRUE;
			bError := FALSE;
			nErrId := 0;
			(* calculate the required source buffer byte size *)
			cbWLen   := nQuantity * 2;
			(* check source buffer and temp buffer length *)
			IF( cbWLen <= cbLength ) AND ( cbWLen <= SIZEOF( stMBWrite.arrBuffer ) ) THEN
				(* prepare request params *)
				stMBWrite.nPort    := nTCPport;
				stMBWrite.nUnitId := nUnitId;
				stMBWrite.arrIpAddr := F_GetIPAddrFromStr( sIPAddr );
				(* copy new reg values to temp buffer *)
				MEMCPY( ADR( stMBWrite.arrBuffer ), pSrcAddr, cbWLen );
				(* reset fb *)
				fbAdsWrite( WRITE := FALSE );
				(* start command execution *)
				fbAdsWrite(IDXGRP :=  DWORD_TO_UDINT(INT_TO_DWORD(MBFCT_WRITEREGISTERS) OR MBADS_IGR_UDP_FLAG),
							IDXOFFS := DWORD_TO_UDINT( SHL( WORD_TO_DWORD( nMBAddr ), 16 ) OR nQuantity ),
							LEN := cbWLen + SIZEOF( stMBWrite.arrIpAddr ) + SIZEOF( stMBWrite.nPort )+ SIZEOF( stMBWrite.nUnitId ),
							SRCADDR := ADR( stMBWrite ), WRITE := TRUE, TMOUT := tTimeout );
				(* go to the wait state *)
				state := 1;
			ELSE
				bBusy := FALSE;
				bError:= TRUE;
				nErrId := 16#702;
			END_IF
		END_IF
	1:(* wait until fb not busy *)
		fbAdsWrite( WRITE := FALSE, BUSY=>bBusy, ERR=>bError, ERRID=>nErrID );
		IF NOT fbAdsWrite.BUSY THEN
			state := 0;
		END_IF
END_CASE
END_FUNCTION_BLOCK

(* POU FB_MBUdpWriteSingleCoil, ST *)
FUNCTION_BLOCK FB_MBUdpWriteSingleCoil
(* Write single digital output (coil, bit access) *)
VAR_INPUT
	sIPAddr	 		: STRING(15);(* IPv4 address of the target device *)
	nTCPPort			: UINT:= MODBUS_TCP_PORT;(* Port number of the target device *)
	nUnitID			: BYTE:=16#FF;(* Identification number of a serial sub-network device *)
	nMBAddr			: WORD;(* Coil address (data bit offset ) *)
	nValue				: WORD;(* New coil value (16#FF00 switches the output on, 16#0000 switches it off) *)
	bExecute			: BOOL;(* Rising edge at this input starts command execution *)
	tTimeout			: TIME:=T#1s;
END_VAR
VAR_OUTPUT
	bBusy				: BOOL;
	bError				: BOOL;
	nErrId				: UDINT;
END_VAR
{library private}
VAR
	state 				: UDINT;
	RisingEdge		: R_TRIG;
	fbAdsWrite			: ADSWRITE := ( NETID := '', PORT := AMSPORT_R3_MODBUSSERV );
	stMBWrite			: ST_MBWriteSingle;
END_VAR
RisingEdge( CLK:= bExecute );
CASE state OF
	0:
		IF RisingEdge.Q THEN
			(* reset outputs *)
			bBusy := TRUE;
			bError := FALSE;
			nErrId := 0;
			(* prepare request params *)
			stMBWrite.nPort    := nTCPport;
			stMBWrite.nUnitId := nUnitId;
			stMBWrite.arrIpAddr := F_GetIPAddrFromStr( sIPAddr );
			(* copy new coil value (2 byte) *)
			MEMCPY(ADR( stMBWrite.nValue ), ADR( nValue ), SIZEOF( stMBWrite.nValue ) );
			(* reset fb *)
			fbAdsWrite( WRITE := FALSE );
			(* start command execution *)
			fbAdsWrite( IDXGRP :=  DWORD_TO_UDINT(INT_TO_DWORD(MBFCT_WRITESINGLECOIL) OR MBADS_IGR_UDP_FLAG),
						IDXOFFS := DWORD_TO_UDINT( SHL( WORD_TO_DWORD( nMBAddr ), 16 ) ),
						LEN := SIZEOF( nValue ) + SIZEOF( stMBWrite.arrIpAddr ) + SIZEOF( stMBWrite.nPort ) + SIZEOF( stMBWrite.nUnitId ),
						SRCADDR := ADR( stMBWrite ), WRITE := TRUE, TMOUT := tTimeout );
			(* go to the wait state *)
			state := 1;
		END_IF
	1:(* wait until fb not busy *)
		fbAdsWrite( WRITE := FALSE, BUSY=>bBusy, ERR=>bError, ERRID=>nErrID );
		IF NOT fbAdsWrite.BUSY THEN
			state := 0;
		END_IF
END_CASE
END_FUNCTION_BLOCK

(* POU FB_MBUdpWriteSingleReg, ST *)
FUNCTION_BLOCK FB_MBUdpWriteSingleReg
(* Write single output register (word access) *)
VAR_INPUT
	sIPAddr	 		: STRING(15);(* IPv4 address of the target device *)
	nTCPPort			: UINT:= MODBUS_TCP_PORT;(* Port number of the target device *)
	nUnitID			: BYTE:=16#FF;(* Identification number of a serial sub-network device *)
	nMBAddr			: WORD;(* Register address (data word offset) *)
	nValue				: WORD;(* New register value (16 bit) *)
	bExecute			: BOOL;(* Rising edge at this input starts command execution *)
	tTimeout			: TIME:=T#1s;
END_VAR
VAR_OUTPUT
	bBusy				: BOOL;
	bError				: BOOL;
	nErrId				: UDINT;
END_VAR
{library private}
VAR
	state 				: UDINT;
	RisingEdge		: R_TRIG;
	fbAdsWrite			: ADSWRITE := ( NETID := '', PORT := AMSPORT_R3_MODBUSSERV );
	stMBWrite			: ST_MBWriteSingle;
END_VAR
RisingEdge( CLK:= bExecute );
CASE state OF
	0:
		IF RisingEdge.Q THEN
			(* reset outputs *)
			bBusy := TRUE;
			bError := FALSE;
			nErrId := 0;
			(* prepare request params *)
			stMBWrite.nPort    := nTCPport;
			stMBWrite.nUnitId := nUnitId;
			stMBWrite.arrIpAddr := F_GetIPAddrFromStr( sIPAddr );
			(* copy new register value (2 bytes) *)
			MEMCPY( ADR( stMBWrite.nValue ), ADR( nValue ), SIZEOF( stMBWrite.nValue ) );
			(* reset fb *)
			fbAdsWrite( WRITE := FALSE );
			(* start command execution *)
			fbAdsWrite( IDXGRP :=  DWORD_TO_UDINT(INT_TO_DWORD(MBFCT_WRITESINGLEREGISTER) OR MBADS_IGR_UDP_FLAG),
						IDXOFFS := DWORD_TO_UDINT( SHL( WORD_TO_DWORD( nMBAddr ), 16 ) ),
						LEN := SIZEOF( nValue ) + SIZEOF( stMBWrite.arrIpAddr ) + SIZEOF( stMBWrite.nPort ) + SIZEOF( stMBWrite.nUnitId ),
						SRCADDR := ADR( stMBWrite ), WRITE := TRUE, TMOUT := tTimeout );
			(* go to the wait state *)
			state := 1;
		END_IF
	1:(* wait until fb not busy *)
		fbAdsWrite( WRITE := FALSE, BUSY=>bBusy, ERR=>bError, ERRID=>nErrID);
		IF NOT fbAdsWrite.BUSY THEN
			state := 0;
		END_IF
END_CASE
END_FUNCTION_BLOCK

(* POU FB_MBWriteCoils, ST *)
FUNCTION_BLOCK FB_MBWriteCoils
(* Write 1..2048 digital outputs (coils, bit access) *)
VAR_INPUT
	sIPAddr	 		: STRING(15);(* IPv4 address of the target device *)
	nTCPPort			: UINT:= MODBUS_TCP_PORT;(* Port number of the target device *)
	nUnitID			: BYTE:=16#FF;(* Identification number of a serial sub-network device *)
	nQuantity			: WORD;(* Number of coils to write (data bits) *)
	nMBAddr			: WORD;(* Address of start coil (data bit offset) *)
	cbLength			: UDINT;(* Max. byte size of source buffer *)
	pSrcAddr			: UDINT;(* Pointer to source buffer *)
	bExecute			: BOOL;(* Rising edge at this input starts command execution *)
	tTimeout			: TIME:=T#1s;
END_VAR
VAR_OUTPUT
	bBusy				: BOOL;
	bError				: BOOL;
	nErrId				: UDINT;
END_VAR
{library private}
VAR
	state 				: UDINT;
	RisingEdge		: R_TRIG;
	fbAdsWrite			: ADSWRITE := ( NETID := '', PORT := AMSPORT_R3_MODBUSSERV, IDXGRP := MBFCT_WRITECOILS );
	stMBWrite			: ST_MBWrite;
	cbWLen			: UDINT;
END_VAR
RisingEdge( CLK:= bExecute );
CASE state OF
	0:
		IF RisingEdge.Q THEN
			(* reset outputs *)
			bBusy := TRUE;
			bError := FALSE;
			nErrId := 0;
			(* calculate the required source buffer byte size *)
			cbWLen   := ( nQuantity + 7 ) / 8;
			(* check source buffer and temp buffer length *)
			IF( cbWLen <= cbLength ) AND ( cbWLen <= SIZEOF( stMBWrite.arrBuffer ) ) THEN
				(* prepare request params *)
				stMBWrite.nPort    := nTCPport;
				stMBWrite.nUnitId := nUnitId;
				stMBWrite.arrIpAddr := F_GetIPAddrFromStr( sIPAddr );
				(* copy new coil values to temp buffer *)
				MEMCPY(ADR(stMBWrite.arrBuffer),pSrcAddr, cbWLen );
				(* reset fb *)
				fbAdsWrite( WRITE := FALSE );
				(* start command execution *)
				fbAdsWrite( IDXOFFS := DWORD_TO_UDINT( SHL( WORD_TO_DWORD( nMBAddr ), 16 ) OR nQuantity ),
							LEN := cbWLen + SIZEOF( stMBWrite.arrIpAddr ) + SIZEOF( stMBWrite.nPort ) + SIZEOF( stMBWrite.nUnitId ),
							SRCADDR := ADR( stMBWrite ), WRITE := TRUE, TMOUT := tTimeout );
				(* go to the wait state *)
				state := 1;
			ELSE
				bBusy := FALSE;
				bError:= TRUE;
				nErrId := 16#702;
			END_IF
		END_IF
	1:(* wait until fb not busy *)
		fbAdsWrite( WRITE := FALSE, BUSY=>bBusy, ERR=>bError, ERRID=>nErrID );
		IF NOT fbAdsWrite.BUSY THEN
			state := 0;
		END_IF
END_CASE
END_FUNCTION_BLOCK

(* POU FB_MBWriteRegs, ST *)
FUNCTION_BLOCK FB_MBWriteRegs
(* Write 1..128 output registers (word access) *)
VAR_INPUT
	sIPAddr	 		: STRING(15);(* IPv4 address of the target device *)
	nTCPPort			: UINT:= MODBUS_TCP_PORT;(* Port number of the target device *)
	nUnitID			: BYTE:=16#FF;(* Identification number of a serial sub-network device *)
	nQuantity			: WORD;(* Number of registers to write (data words) *)
	nMBAddr			: WORD;(* Address of start register (data word offset) *)
	cbLength			: UDINT;(* Max. byte size of source buffer *)
	pSrcAddr			: UDINT;(* Pointer to source buffer *)
	bExecute			: BOOL;(* Rising edge at this input starts command execution *)
	tTimeout			: TIME:=T#1s;
END_VAR
VAR_OUTPUT
	bBusy				: BOOL;
	bError				: BOOL;
	nErrId				: UDINT;
END_VAR
{library private}
VAR
	state 				: UDINT;
	RisingEdge		: R_TRIG;
	fbAdsWrite			: ADSWRITE := ( NETID := '', PORT := AMSPORT_R3_MODBUSSERV, IDXGRP := MBFCT_WRITEREGISTERS );
	stMBWrite			: ST_MBWrite;
	cbWLen			: UDINT;
END_VAR
RisingEdge( CLK:= bExecute );
CASE state OF
	0:
		IF RisingEdge.Q THEN
			(* reset outputs *)
			bBusy := TRUE;
			bError := FALSE;
			nErrId := 0;
			(* calculate the required source buffer byte size *)
			cbWLen   := nQuantity * 2;
			(* check source buffer and temp buffer length *)
			IF( cbWLen <= cbLength ) AND ( cbWLen <= SIZEOF( stMBWrite.arrBuffer ) ) THEN
				(* prepare request params *)
				stMBWrite.nPort    := nTCPport;
				stMBWrite.nUnitId := nUnitId;
				stMBWrite.arrIpAddr := F_GetIPAddrFromStr( sIPAddr );
				(* copy new reg values to temp buffer *)
				MEMCPY( ADR( stMBWrite.arrBuffer ), pSrcAddr, cbWLen );
				(* reset fb *)
				fbAdsWrite( WRITE := FALSE );
				(* start command execution *)
				fbAdsWrite( IDXOFFS := DWORD_TO_UDINT( SHL( WORD_TO_DWORD( nMBAddr ), 16 ) OR nQuantity ),
							LEN := cbWLen + SIZEOF( stMBWrite.arrIpAddr ) + SIZEOF( stMBWrite.nPort )+ SIZEOF( stMBWrite.nUnitId ),
							SRCADDR := ADR( stMBWrite ), WRITE := TRUE, TMOUT := tTimeout );
				(* go to the wait state *)
				state := 1;
			ELSE
				bBusy := FALSE;
				bError:= TRUE;
				nErrId := 16#702;
			END_IF
		END_IF
	1:(* wait until fb not busy *)
		fbAdsWrite( WRITE := FALSE, BUSY=>bBusy, ERR=>bError, ERRID=>nErrID );
		IF NOT fbAdsWrite.BUSY THEN
			state := 0;
		END_IF
END_CASE
END_FUNCTION_BLOCK

(* POU FB_MBWriteSingleCoil, ST *)
FUNCTION_BLOCK FB_MBWriteSingleCoil
(* Write single digital output (coil, bit access) *)
VAR_INPUT
	sIPAddr	 		: STRING(15);(* IPv4 address of the target device *)
	nTCPPort			: UINT:= MODBUS_TCP_PORT;(* Port number of the target device *)
	nUnitID			: BYTE:=16#FF;(* Identification number of a serial sub-network device *)
	nMBAddr			: WORD;(* Coil address (data bit offset ) *)
	nValue				: WORD;(* New coil value (16#FF00 switches the output on, 16#0000 switches it off) *)
	bExecute			: BOOL;(* Rising edge at this input starts command execution *)
	tTimeout			: TIME:=T#1s;
END_VAR
VAR_OUTPUT
	bBusy				: BOOL;
	bError				: BOOL;
	nErrId				: UDINT;
END_VAR
{library private}
VAR
	state 				: UDINT;
	RisingEdge		: R_TRIG;
	fbAdsWrite			: ADSWRITE := ( NETID := '', PORT := AMSPORT_R3_MODBUSSERV, IDXGRP := MBFCT_WRITESINGLECOIL );
	stMBWrite			: ST_MBWriteSingle;
END_VAR
RisingEdge( CLK:= bExecute );
CASE state OF
	0:
		IF RisingEdge.Q THEN
			(* reset outputs *)
			bBusy := TRUE;
			bError := FALSE;
			nErrId := 0;
			(* prepare request params *)
			stMBWrite.nPort    := nTCPport;
			stMBWrite.nUnitId := nUnitId;
			stMBWrite.arrIpAddr := F_GetIPAddrFromStr( sIPAddr );
			(* copy new coil value (2 byte) *)
			MEMCPY(ADR( stMBWrite.nValue ), ADR( nValue ), SIZEOF( stMBWrite.nValue ) );
			(* reset fb *)
			fbAdsWrite( WRITE := FALSE );
			(* start command execution *)
			fbAdsWrite( IDXOFFS := DWORD_TO_UDINT( SHL( WORD_TO_DWORD( nMBAddr ), 16 ) ),
						LEN := SIZEOF( nValue ) + SIZEOF( stMBWrite.arrIpAddr ) + SIZEOF( stMBWrite.nPort ) + SIZEOF( stMBWrite.nUnitId ),
						SRCADDR := ADR( stMBWrite ), WRITE := TRUE, TMOUT := tTimeout );
			(* go to the wait state *)
			state := 1;
		END_IF
	1:(* wait until fb not busy *)
		fbAdsWrite( WRITE := FALSE, BUSY=>bBusy, ERR=>bError, ERRID=>nErrID );
		IF NOT fbAdsWrite.BUSY THEN
			state := 0;
		END_IF
END_CASE
END_FUNCTION_BLOCK

(* POU FB_MBWriteSingleReg, ST *)
FUNCTION_BLOCK FB_MBWriteSingleReg
(* Write single output register (word access) *)
VAR_INPUT
	sIPAddr	 		: STRING(15);(* IPv4 address of the target device *)
	nTCPPort			: UINT:= MODBUS_TCP_PORT;(* Port number of the target device *)
	nUnitID			: BYTE:=16#FF;(* Identification number of a serial sub-network device *)
	nMBAddr			: WORD;(* Register address (data word offset) *)
	nValue				: WORD;(* New register value (16 bit) *)
	bExecute			: BOOL;(* Rising edge at this input starts command execution *)
	tTimeout			: TIME:=T#1s;
END_VAR
VAR_OUTPUT
	bBusy				: BOOL;
	bError				: BOOL;
	nErrId				: UDINT;
END_VAR
{library private}
VAR
	state 				: UDINT;
	RisingEdge		: R_TRIG;
	fbAdsWrite			: ADSWRITE := ( NETID := '', PORT := AMSPORT_R3_MODBUSSERV, IDXGRP := MBFCT_WRITESINGLEREGISTER );
	stMBWrite			: ST_MBWriteSingle;
END_VAR
RisingEdge( CLK:= bExecute );
CASE state OF
	0:
		IF RisingEdge.Q THEN
			(* reset outputs *)
			bBusy := TRUE;
			bError := FALSE;
			nErrId := 0;
			(* prepare request params *)
			stMBWrite.nPort    := nTCPport;
			stMBWrite.nUnitId := nUnitId;
			stMBWrite.arrIpAddr := F_GetIPAddrFromStr( sIPAddr );
			(* copy new register value (2 bytes) *)
			MEMCPY( ADR( stMBWrite.nValue ), ADR( nValue ), SIZEOF( stMBWrite.nValue ) );
			(* reset fb *)
			fbAdsWrite( WRITE := FALSE );
			(* start command execution *)
			fbAdsWrite( IDXOFFS := DWORD_TO_UDINT( SHL( WORD_TO_DWORD( nMBAddr ), 16 ) ),
						LEN := SIZEOF( nValue ) + SIZEOF( stMBWrite.arrIpAddr ) + SIZEOF( stMBWrite.nPort ) + SIZEOF( stMBWrite.nUnitId ),
						SRCADDR := ADR( stMBWrite ), WRITE := TRUE, TMOUT := tTimeout );
			(* go to the wait state *)
			state := 1;
		END_IF
	1:(* wait until fb not busy *)
		fbAdsWrite( WRITE := FALSE, BUSY=>bBusy, ERR=>bError, ERRID=>nErrID);
		IF NOT fbAdsWrite.BUSY THEN
			state := 0;
		END_IF
END_CASE
END_FUNCTION_BLOCK
